INTERFACE IPLCOpenBase

PROPERTY Busy : BOOL
GET
END_GET
END_PROPERTY

PROPERTY ConsumeDone : Bool
GET
END_GET
END_PROPERTY

PROPERTY Done : BOOL
GET
END_GET
END_PROPERTY

PROPERTY Error : BOOL
GET
END_GET
END_PROPERTY

END_INTERFACE

(* stored: Version 1.1.0.1, ProductVersion 3.1.4024.12
   Itf IPLCOpenBase: Id {30663370-63aa-4ece-9d78-1fee533d169f}
   Property Busy: Id {dbad1434-9112-4a9a-ac6b-cefc61b97ffa}
   Get Get: Id {a8b28f5c-70eb-4c8c-96af-d12c10b903a3}
   Property ConsumeDone: Id {90e95edf-6f37-4b47-a3c8-0e660f477518}
   Get Get: Id {a39141f9-422e-43a8-aea4-15c7a351e21c}
   Property Done: Id {75bee3fb-619b-4a49-8989-a90772baef00}
   Get Get: Id {77fd2a6c-b610-4aa9-845d-bc5bb1f8df12}
   Property Error: Id {70e9ec0c-ad6f-4119-acdc-0be5d3930437}
   Get Get: Id {a51bc305-8a6e-4d61-970b-4293ab47c457} *)
